// TIA Portal V20 export
// export: Created 2025-12-01T14:57:14.5479989Z, ExportSetting None, DisplayName Totally Integrated Automation Portal, DisplayVersion V20 Update 3, DisplayName TIA Portal Openness, DisplayVersion V20 Update 3, DisplayName TIA Portal Version Control Interface, DisplayVersion V20 Update 3, DisplayName STEP 7 Professional, DisplayVersion V20 Update 3, DisplayName STEP 7 Safety, DisplayVersion V20 Update 2, DisplayName WinCC Basic/Comfort/Advanced, DisplayVersion V20 Update 3, DisplayName WinCC Professional, DisplayVersion V20 Update 3, DisplayName WinCC Unified, DisplayVersion V20 Update 3
FUNCTION "FC800_JDT01ControlTracking" : Void   // FC800, LAD
{ S7_Optimized_Access := 'FALSE' }
AUTHOR : TRACKING
NAME : 20141014
VERSION : 4.0
// stored: AutoNumber false, SetENOAutomatically false
BEGIN

NETWORK
TITLE = Previo
// -----------------------------------------------------------------------
// --- Inicialializacion
// --- Borrado de la Base de Datos

      CALL  "FC801_JDT01ControlCOM";  // Control del Puerto
      CALL  "FC806_JDT01Borrado";



NETWORK
TITLE = Distribucion Dependiendo del Tipo de JDT
///////////////////////////////////////////////////////////////////////////
///////////////////////////////////////////////////////////////////////////
///////////////////////////////////////////////////////////////////////////
/// --- Distribucion Dependiendo del Tipo de JDT (ACTUAL o VIEJO)
      SET;
      A     "Activar_JdTAntiguo";
      JC    Agencia_TrackingViejo;
      JU    Agencia_TrackingActual;



NETWORK
TITLE = Control del Sistema >>> Agencia de TRACKING ACTUAL
///////////////////////////////////////////////////////////////////////////
///////////////////////////////////////////////////////////////////////////
///////////////////////////////////////////////////////////////////////////
/// --- Agencia de TRACKING ACTUAL
Agencia_TrackingActual:NOP   0;

// ---------------------------------------------------------------------
// --- Control de Recepcion de Eventos

      CALL  "FC802_JDT01RecJdTMensaje";
      CALL  "FC804_JDT01AnalisisRecibidos";
      CALL  "FC810_EventosRecibidos"
      ( NumJDT := 1
      );

      CALL  "FC823_OrdenesMesas";
      CALL  "FC821_OrdenesDispositivos";

// ---------------------------------------------------------------------
// --- Control de EmisionEventos de Eventos


      CALL  "FC811_EventosGenerados"
      ( NumJdT := 1
      );
      CALL  "FC805_JDT01AnalisisEnviados";
      CALL  "FC803_JDT01EmiJdTMensaje";

      CALL  "FC822_EstadosMesas";
      CALL  "FC820_EstadosDispositivos";


// ---------------------------------------------------------------------
// --- Control de EmisionEventos de Router
//     *  Proceso Inicialización bucle
//     *  Eventos de la Pantalla (Movimientos)
//     *  Eventos de Reset V2.0   >>> 2023 01 05

//      CALL  "FC816_EventosEnv_Router"
//         NumJDT :=1


// NIEVES 10/04/25
      CALL  "FC717_Emision_Routing"
      ( NumJDT := 1
      );

      CALL  "FC815_EventosEnv_Control"
      ( NumJDT := 1
      );
      CALL  "FC817_EventosEnv_Reset"
      ( NumJDT := 1
      );


///////////////////////////////////////////////////////////////////////////
      JU    Fin;



NETWORK
TITLE = Control del Sistema >>> Agencia de TRACKING VIEJO
///////////////////////////////////////////////////////////////////////////
///////////////////////////////////////////////////////////////////////////
///////////////////////////////////////////////////////////////////////////
/// --- Agencia de TRACKING ACTUAL
Agencia_TrackingViejo:NOP   0;

///////////////////////////////////////////////////////////////////////////
// --- Control de Recepcion de Eventos

      CALL  "FC821_OrdenesDispositivos";


///////////////////////////////////////////////////////////////////////////
// --- Control de EmisionEventos de Eventos

      CALL  "FC811_EventosGenerados"
      ( NumJdT := 1
      );
      CALL  "FC805_JDT01AnalisisEnviados";

      CALL  "FC820_EstadosDispositivos";


///////////////////////////////////////////////////////////////////////////
      JU    Fin;



NETWORK
TITLE = Final de la Funcion
///////////////////////////////////////////////////////////////////////////
///////////////////////////////////////////////////////////////////////////
///////////////////////////////////////////////////////////////////////////
/// --- Final de la Funcion
Fin:  NOP   0;


END_FUNCTION
